METHOD line_line_angle : bool
VAR_INPUT
	p0:sc_pnt;
	p1:sc_pnt;
	p2:sc_pnt;
	angle_deg:REFERENCE TO LREAL;
END_VAR
VAR
	p00,p11,p22,v1,v2:Vector_3;
	dot,angle_rad:LREAL;
END_VAR
p00:=p_to_v(p0);
p11:=p_to_v(p1);
p22:=p_to_v(p2);

v1:=V3_SUB(p00,p11);
v2:=V3_SUB(p22,p11);

v1:=V3_NORMALIZED(v1);
v2:=V3_NORMALIZED(v2);

dot:=V3_DOT(v1,v2);
angle_rad:=ACOS(dot);
angle_deg:=angle_rad*to_degrees;
END_METHOD

METHOD arc_line_angle : bool
VAR_INPUT
	p0:sc_pnt;
	p1:sc_pnt;
	p2:sc_pnt;
	p3:sc_pnt;
	angle_deg:REFERENCE TO LREAL;
END_VAR
VAR
	pi:sc_pnt;

END_VAR
interpolate_arc(p0,p1,p2,0.9,pi);
line_line_angle(pi,p2,p3,angle_deg);
END_METHOD

METHOD p_to_v : Vector_3 //sc_pnt to vector3
VAR_INPUT
	in:sc_pnt;
END_VAR
p_to_v.x:=in.x;
p_to_v.y:=in.y;
p_to_v.z:=in.z;
END_METHOD

METHOD get_blockangles : BOOL
VAR_INPUT
	blockvec:REFERENCE TO vector_sc_segment;
	start:REFERENCE TO UDINT;
	end:REFERENCE TO UDINT;
END_VAR
VAR	
	i: UDINT;
	angle_deg:LREAL;
END_VAR
IF(blockvec.size()>0)THEN //! Vector safe.}
	
	FOR i:=start TO end-1 DO
		
		IF(blockvec.data[i].primitive_id=sc_primitive_id.line AND  blockvec.data[i+1].primitive_id=sc_primitive_id.line)THEN
			line_line_angle(blockvec.data[i].pnt_s,blockvec.data[i].pnt_e,blockvec.data[i+1].pnt_e,angle_deg);
			blockvec.data[i].angle_end:=angle_deg;
		END_IF
		
		IF(blockvec.data[i].primitive_id=sc_primitive_id.line AND (blockvec.data[i+1].primitive_id=sc_primitive_id.arc_ccw OR blockvec.data[i+1].primitive_id=sc_primitive_id.arc_cw))THEN
			line_arc_angle(blockvec.data[i].pnt_s,blockvec.data[i].pnt_e,blockvec.data[i+1].pnt_c,blockvec.data[i+1].pnt_e,angle_deg);
			blockvec.data[i].angle_end:=angle_deg;
		END_IF
		
		IF((blockvec.data[i].primitive_id=sc_primitive_id.arc_ccw OR blockvec.data[i].primitive_id=sc_primitive_id.arc_cw) AND blockvec.data[i+1].primitive_id=sc_primitive_id.line)THEN
			arc_line_angle(blockvec.data[i].pnt_s,blockvec.data[i].pnt_c,blockvec.data[i].pnt_e,blockvec.data[i+1].pnt_e,angle_deg);
			blockvec.data[i].angle_end:=angle_deg;
		END_IF
		
		IF((blockvec.data[i].primitive_id=sc_primitive_id.arc_ccw OR blockvec.data[i].primitive_id=sc_primitive_id.arc_cw) AND (blockvec.data[i+1].primitive_id=sc_primitive_id.arc_ccw OR blockvec.data[i+1].primitive_id=sc_primitive_id.arc_cw))THEN
			arc_arc_angle(blockvec.data[i].pnt_s,blockvec.data[i].pnt_c,blockvec.data[i].pnt_e,blockvec.data[i+1].pnt_c,blockvec.data[i+1].pnt_e,angle_deg);
			blockvec.data[i].angle_end:=angle_deg;
		END_IF
	END_FOR
END_IF
END_METHOD

METHOD get_corner_ve_blockangles : BOOL
VAR_INPUT
	blockvec:REFERENCE TO vector_sc_segment;
	start:REFERENCE TO UDINT;
	end:REFERENCE TO UDINT;
END_VAR
VAR	
	i: UDINT;
	angle_deg,factor,ve:LREAL;
END_VAR
IF(blockvec.size()<>0)THEN
	FOR i:=start TO  end-1 DO
		
		IF(blockvec.data[i].angle_end<=STOP_ANGLE)THEN //! Stop required.
			blockvec.data[i].vel_end:=0;
			//! Set next block vo to zero.
			IF(i<blockvec.size()-1)THEN
				blockvec.data[i+1].vel_start:=0;
			END_IF
		END_IF
	
		IF(blockvec.data[i].angle_end>STOP_ANGLE)THEN //! Percentage ve up to 180 degrees. //! 180 degrees = colinear.
			angle_deg:=blockvec.data[i].angle_end;
			factor:=(angle_deg-STOP_ANGLE)/STOP_ANGLE; //! 0-1, 1=straight on. 0=90 degrees.
			ve:=blockvec.data[i].vel_max*factor*ANGLE_VEL_FACTOR;
	
			blockvec.data[i].vel_end:=ve;
			//! Set next block vo to this ve.
			IF(i<blockvec.size()-1)THEN
				blockvec.data[i+1].vel_start:=ve;
			END_IF
		END_IF
		
	END_FOR
END_IF
END_METHOD

METHOD sc_get_gforce : bool
VAR_INPUT
	vel_mm_sec:LREAL;
	radius:LREAL;
	gforce:LREAL;
END_VAR
VAR	
	circumfence: LREAL;
	rps: LREAL;
	a:LREAL;
END_VAR
circumfence:=(radius*2)*M_PI;
rps:=vel_mm_sec/circumfence;
a:=4*(M_PI*M_PI)*radius*(rps*rps); //! [mm/s^2]
gforce:=a*0.0001; //! [g]
END_METHOD

METHOD get_velmax_gforce : bool
VAR_INPUT
	blockvec:REFERENCE TO vector_sc_segment;
	gforcemax:LREAL;
	start:REFERENCE TO UDINT;
	end:REFERENCE TO UDINT;
END_VAR
VAR
	i:UDINT;
	radius,gforce,maxvel_arc:LREAL;
	vm:LREAL;
END_VAR
IF(blockvec.size()<>0)THEN
	FOR i:=start TO end-1 DO
		IF(blockvec.data[i].primitive_id=sc_primitive_id.arc_cw OR blockvec.data[i].primitive_id=sc_primitive_id.arc_ccw)THEN	
			
			radius:=blockvec.data[i].radius;	
			
			//! Checks gforce using the program's velmax value.	
			vm:=blockvec.data[i].vel_max;							
			sc_get_gforce(vm,radius,gforce);
	
			IF(gforce>gforcemax)THEN
				maxvel_arc:=0;
				sc_set_gforce(radius,gforcemax,maxvel_arc);
				blockvec.data[i].vel_max:=maxvel_arc;
			END_IF			
		END_IF
	END_FOR
END_IF
END_METHOD

METHOD sc_optimize_all : BOOL
VAR_INPUT
	blockvec:REFERENCE TO vector_sc_segment;
	line_start:UDINT;
	line_end:UDINT;
END_VAR
line_start:=LIMIT(0,line_start,blockvec.size());
line_end:=LIMIT(line_start,line_end,blockvec.size());



//! Calculate motion block corners.
get_blockangles(blockvec,line_start,line_end);

//! Set end velocity, based on block corners, if no angle, ve is set to vm at this stage.
get_corner_ve_blockangles(blockvec,line_start,line_end);

//! Set the velmax for arc's using gforce value. Set the velmax for lines to program velmax.
get_velmax_gforce(blockvec,gforcemax,line_start,line_end);

//set g0 ve vo
sc_optimize_G0_ve(blockvec,line_start,line_end);

//optimize ve <--
sc_optimize_G123_ve_backward(blockvec,line_start,line_end);

//optimize ve -->
sc_optimize_G123_ve_forward(blockvec,line_start,line_end);
END_METHOD

METHOD sc_optimize_G0_ve : BOOL
VAR_INPUT
	blockvec:REFERENCE TO vector_sc_segment;
	start:REFERENCE TO UDINT;
	end:REFERENCE TO UDINT;
END_VAR
VAR
	i:UDINT;
END_VAR
IF(blockvec.size()<>0)THEN
	FOR i:=start TO end-1 DO
	
		//! End velocity=0 if motion is G0, rapid.
		IF(blockvec.data[i].primitive_id=sc_primitive_id.rapid)THEN 
			blockvec.data[i].vel_start:=0;
			blockvec.data[i].vel_end:=0;
	
			//! Set next block vo to 0.
			IF(i<blockvec.size()-1)THEN
				blockvec.data[i+1].vel_start:=0;
			END_IF
		END_IF
	END_FOR
END_IF
END_METHOD

METHOD sc_optimize_G123_ve_backward :BOOL
VAR_INPUT
	blockvec:REFERENCE TO vector_sc_segment;
	start:REFERENCE TO UDINT;
	end:REFERENCE TO UDINT;
END_VAR
VAR
	i:UDINT;
	vo,ve,vm,tarpos:LREAL;
	r_vel,r_acc,r_pos:LREAL;
	finish:BOOL;
	p_data:sc_data;
	pcurve:sc_engine;
	j:LREAL;
	
END_VAR
IF(blockvec.size()<>0)THEN
	FOR i:=end-1 TO start+1 BY-1 DO 
		
		IF(blockvec.data[i].primitive_id<>sc_primitive_id.rapid AND blockvec.data[i].primitive_id<>sc_primitive_id.empty)THEN 
			//! Swap vo,ve.
			ve:=blockvec.data[i].vel_start;
			vo:=blockvec.data[i].vel_end;
			vm:=blockvec.data[i].vel_max;
			tarpos:=blockvec.data[i].path_lenght;	

			MEMUtils.MemSet(ADR(p_data),0,SIZEOF(p_data));
			
			pcurve.set_cycle_time(CT,p_data);
			
			finish:=FALSE;
			WHILE NOT finish DO				
				pcurve.set_data(tarpos,vo,ve,vm,limits.max_acc,limits.max_jerk,1,p_data);	
				pcurve.update(p_data,1);
				pcurve.get_result(r_pos,r_vel,r_acc,finish,p_data);			
			END_WHILE
			
			IF(ve<>0)THEN
				blockvec.data[i].vel_start:=r_vel;
				blockvec.data[i-1].vel_end:=r_vel;
			END_IF
			
			blockvec.data[i].back_optim:=TRUE;
		END_IF
	END_FOR
END_IF
END_METHOD

METHOD sc_optimize_G123_ve_forward : BOOL
VAR_INPUT
	blockvec:REFERENCE TO vector_sc_segment;
	start:REFERENCE TO UDINT;
	end:REFERENCE TO UDINT;
END_VAR
VAR
	i:UDINT;
	vo,ve,vm,tarpos:LREAL;
	r_vel,r_acc,r_pos:LREAL;
	finish:BOOL;
	p_data:sc_data;
	pcurve:sc_engine;

END_VAR
IF(blockvec.size()<>0)THEN	
	FOR i:=start TO end-1 DO 
	
		IF(blockvec.data[i].primitive_id<>sc_primitive_id.rapid AND blockvec.data[i].primitive_id<>sc_primitive_id.empty)THEN 
	
			vo:=blockvec.data[i].vel_start;
			ve:=blockvec.data[i].vel_end;
			vm:=blockvec.data[i].vel_max;
			tarpos:=blockvec.data[i].path_lenght;
			
			MEMUtils.MemSet(ADR(p_data),0,SIZEOF(p_data));
			
			pcurve.set_cycle_time(CT,p_data);
						
			finish:=FALSE;
			WHILE NOT finish DO			
				pcurve.set_data(tarpos,vo,ve,vm,limits.max_acc,limits.max_jerk,1,p_data);	
				pcurve.update(p_data,1);
				pcurve.get_result(r_pos,r_vel,r_acc,finish,p_data);
			END_WHILE
			
			IF(ve<>0)THEN
				blockvec.data[i].vel_end:=r_vel;		
				IF(i<blockvec.size()-1)THEN  
					blockvec.data[i+1].vel_start:=r_vel;
				END_IF				
			END_IF
			
			blockvec.data[i].forward_optim:=TRUE;
		END_IF
	END_FOR
END_IF
END_METHOD

METHOD sc_set_gforce : bool
VAR_INPUT
	radius:LREAL;
	gforce:LREAL;
	vel_mm_sec:reference TO LREAL;
END_VAR

VAR
	rps: LREAL;
	circumfence: LREAL;
	a:LREAL;
END_VAR
circumfence:=(radius*2)*M_PI;
a:=gforce/0.0001;
rps:= SQRT(a/(4*(M_PI*M_PI)*radius));
vel_mm_sec:=rps*circumfence;
END_METHOD

METHOD interpolate_lenght
VAR_INPUT
	start,end,progress:LREAL;
	li:REFERENCE TO LREAL;
END_VAR
IF(start<end)THEN
	li:=start+(progress*NETTO(start,end));
	return;
END_IF
IF(start>end)THEN
	li:=start-(progress*NETTO(start,end));
	return;
END_IF
IF(start=end)THEN
	li:=end;
END_IF
END_METHOD

METHOD interpolate_arc
VAR_INPUT
	p1:sc_pnt;//! start position
	p2:sc_pnt;//! end position 
	center:sc_pnt;//! center IJK
	progress:LREAL;
	pi:REFERENCE TO sc_pnt;
END_VAR
VAR
	radius:LREAL;
	circumference:LREAL;
	startingAngle,endingAngle:LREAL;
	chordSquared,tau,chordHeight:LREAL;
	theta:LREAL;
	arcLengthMM:LREAL;
	angleNow:LREAL;

END_VAR
// add center offset IJ
center.x:=center.x+p1.x;
center.y:=center.y+p1.y;
// Compute geometry.
radius:=SQRT(EXPT(center.x-p1.x,2)+EXPT(center.y-p1.y,2)); 
circumference:=2.0*M_PI*radius;
startingAngle:=math.atan2(p1.y-center.y,p1.x-center.x);
endingAngle:=math.atan2(p2.y-center.y,p2.x-center.x);

// Compute chord height of arc.
chordSquared:=SQRT(EXPT(p2.x-p1.x,2)+EXPT(p2.y-p1.y,2));
tau:=SQRT(EXPT(radius,2)-(chordSquared/4));
chordHeight := radius - tau;

// Compute angle between lines.
theta:=endingAngle-startingAngle;

	//COUNTERCLOCKWISE
	IF (theta < 0)THEN
		theta:=theta+2*M_PI;
	END_IF

	//CLOCKWISE
	IF (theta >= 0)THEN	
		theta:=theta-2*M_PI;;
	END_IF


arcLengthMM:=ABS(circumference*(theta/(2*M_PI)));

//rotate point xy interpolate
angleNow:=startingAngle+theta*progress;
pi.x:=radius*COS(angleNow)+center.x;
pi.y:=radius*SIN(angleNow)+center.y;

IF(progress=1)THEN
	pi.x:=p2.x;
	pi.y:=p2.y;
END_IF

//z interpolate
interpolate_lenght(p1.z,p2.z,progress,pi.z);
END_METHOD

METHOD update_motion_and_interpolator : bool
VAR
	
END_VAR
//feed override
IF(pause_request OR stop_request)THEN
	maxvel_fo:=0;
ELSE
	maxvel_fo:=LIMIT(0,feed_override,100)/100;
END_IF


//motion cycle time
motion.set_cycle_time(CT,motion_data);

CASE state OF
	
	program_run://-------------------------------------------------------------------------------------------
	
		//motion
		motion.set_data(p.traject_lenght_end,p.vel_start,p.vel_end,p.vel_max,limits.max_acc,limits.max_jerk,maxvel_fo,motion_data);	
		motion.update(motion_data,0);
		motion.get_result(engine_outpos,velocity,acceleration,engine_finished,motion_data);
		//programmed vel
		programmed_velocity:=p.vel_max;
		
		//line progress
		line_progress:=(engine_outpos-p.traject_lenght_begin)/p.path_lenght;
		IF(FPU.IsLRealNaN(line_progress))THEN
			line_progress:=0;
		END_IF
		
		//interpolation
		IF(p.primitive_id=sc_primitive_id.line OR p.primitive_id=sc_primitive_id.rapid)THEN
			interpolate_line(p.pnt_s,p.pnt_e,line_progress,xyz);
		ELSIF(p.primitive_id=sc_primitive_id.arc_ccw OR p.primitive_id=sc_primitive_id.arc_cw)THEN
			interpolate_arc(p.pnt_s,p.pnt_e,p.pnt_c,line_progress,xyz);
		END_IF
		
	program_jog://-------------------------------------------------------------------------------------------
		
		
		motion.set_jog(jog_cmd.x_up,jog_cmd.x_dn,limits.min_quote_x,limits.max_quote_x,limits.max_vel,limits.max_acc,limits.max_jerk,motion_data);	
		motion.get_result(engine_outpos,velocity,acceleration,engine_finished,motion_data);
		xyz.x:=engine_outpos;
	
		
		
		
END_CASE
END_METHOD

METHOD interpolate_line
VAR_INPUT
	p0:sc_pnt;//! start point
	p1:sc_pnt;//! end pont
	progress:LREAL;
	pi:REFERENCE TO sc_pnt;
END_VAR
interpolate_lenght(p0.x,p1.x,progress,pi.x);
interpolate_lenght(p0.y,p1.y,progress,pi.y);
interpolate_lenght(p0.z,p1.z,progress,pi.z);
END_METHOD

METHOD round : LREAL
VAR_INPUT
	in : LREAL;
	N : INT;
END_VAR
VAR
	X: LREAL;
END_VAR
VAR
	DECADES : ARRAY[0..8] OF LREAL :=[ 1.0,10.0,100.0,1000.0,10000.0,10000.0,100000.0,1000000.0,10000000.0];
END_VAR
X := DECADES[LIMIT(0,N,8)];
ROUND := DINT_TO_LREAL(LREAL_TO_DINT(in * X)) / X;
END_METHOD

METHOD netto : LREAL
VAR_INPUT
	a,b:LREAL;
END_VAR
VAR
	diff_:LREAL;
END_VAR
diff_:=0;
IF(a<0 AND b<0)THEN
	a:=ABS(a);
	b:=ABS(b);
	diff_:=ABS(a-b);
END_IF
IF(a>=0 AND b>=0)THEN
	diff_:=ABS(a-b);
END_IF
IF(a<=0 AND b>=0)THEN
	diff_:=ABS(a)+b;
END_IF
IF(a>=0 AND b<=0)THEN
	diff_:=a+ABS(b);
END_IF
NETTO:=diff_;
END_METHOD

METHOD set_pnt_at : bool
VAR_INPUT
	pnt:REFERENCE TO sc_pnt;
	index:UDINT;
END_VAR
motion_vec.data[index].pnt_s:=pnt;
END_METHOD

END_FUNCTION_BLOCK

// MyController/Application/cnc/vector/functions/vector_at
FUNCTION vector_at : sc_segment
VAR_INPUT
	ptr:REFERENCE TO vector_sc_segment;
	index:UDINT;
END_VAR

IF(index>ptr.size()-1)THEN
	index:=ptr.size()-1;
END_IF
IF(index<0)THEN
	index:=0;
END_IF
vector_at:=ptr.data[index];

END_FUNCTION

// MyController/Application/cnc/vector/vector_sc_segment
FUNCTION_BLOCK vector_sc_segment
VAR_INPUT	
	data:ARRAY[0..MAX_GCODE_LINE+1]OF sc_segment;
END_VAR
VAR_OUTPUT
END_VAR
VAR	
	last_ptr:UDINT;
END_VAR

METHOD clear : bool
VAR_INPUT
END_VAR
VAR
	i:UDINT;
END_VAR
MEMUtils.MemSet(ADR(data),0,SIZEOF(data));
last_ptr:=0;
END_METHOD

METHOD end : UDINT
VAR_INPUT
END_VAR
end:=last_ptr;
END_METHOD

METHOD begin : int
VAR_INPUT
END_VAR
begin:=0;
END_METHOD

METHOD push_back : bool
VAR_INPUT
	in:sc_segment;
END_VAR
MEMUtils.MemCpy(ADR(data[last_ptr]),ADR(in),SIZEOF(in));
last_ptr:=last_ptr+1;
END_METHOD

METHOD back : sc_segment
VAR_INPUT
END_VAR
back:=data[last_ptr-1];
END_METHOD

METHOD front : sc_segment
VAR_INPUT
END_VAR
front:=data[0];
END_METHOD

METHOD size : UDINT
VAR_INPUT
END_VAR
size:=last_ptr;
END_METHOD

METHOD insert : bool
VAR_INPUT
	pos:UDINT;
	vec:REFERENCE TO vector_sc_segment;
END_VAR
VAR
	i:UDINT;
END_VAR
//libero lo spazio spostando avanti i vettori successivi al punto di inserimento
IF(vec.size()>0)THEN
	IF(last_ptr<>0)THEN
		FOR i:=pos TO last_ptr-1 DO
			MEMUtils.MemCpy(ADR(data[i+vec.size()]),ADR(data[i]),SIZEOF(data[i]));
			//data[i+vec.size()]:=data[i];
		END_FOR
		last_ptr:=i+vec.size();
	END_IF


	//copio il nuovo array partendo dalla posizione desiderata
	FOR i:=0 TO vec.size()-1 DO
		MEMUtils.MemCpy(ADR(data[i+pos]),ADR(vec.data[i]),SIZEOF(vec.data[i]));
		//data[i+pos]:=vec.data[i];
		//se non ho inserito prima nessun vettore,avanzo il puntatore alla fine della lunghezza del vettore che copio
		IF(last_ptr=0)THEN
			last_ptr:=i+vec.size();
		END_IF 	
	END_FOR
END_IF
END_METHOD

END_FUNCTION_BLOCK

// MyController/Application/cnc/vector/functions/vector_nr_increment
FUNCTION vector_nr_increment : bool
VAR_INPUT
	ptr:REFERENCE TO vector_sc_segment;
	n:REFERENCE TO UDINT;
END_VAR

n:=n+1;
n:=MIN(n,ptr.size());
n:=MAX(n,0);

END_FUNCTION

// MyController/Application/cnc/motion/sc_engine
FUNCTION_BLOCK sc_engine
VAR_INPUT
END_VAR
VAR_OUTPUT
END_VAR
VAR
END_VAR

METHOD set_data : bool
VAR_INPUT
	ds:LREAL;//target
	vo:LREAL;//begin velocity
	ve:LREAL;//end velocity
	vs:LREAL;//max velocity
	a:LREAL;//acceleration
	gain:LREAL;//0-100
	ovr:LREAL;//override 0-1
	p:REFERENCE TO sc_data;//data structure
END_VAR
//!limit gain
gain:=LIMIT(0.001,gain,100);

ve:=ve*ovr;
vs:=vs*ovr;

IF(vs=0)THEN
	vs:=0.000001;
	p.stop:=TRUE;
END_IF

//target position change
IF(ds<>p.ds_old)THEN
	p.ds:=ds;
	p.ds_old:=p.ds;
	p.init:=TRUE;
END_IF

//max vel change
IF(vs<>p.vs_old)THEN
	p.vs:=vs;
	p.vs_old:=p.vs;
	p.init:=TRUE;
END_IF

p.vo:=vo;
p.vs:=vs;
p.ve:=ve;
p.a:=a;
p.gain:=gain;
END_METHOD

METHOD get_result : bool
VAR_INPUT
	pos:REFERENCE TO LREAL;
	vel:REFERENCE TO LREAL;
	acc:REFERENCE TO LREAL;
	finish:REFERENCE TO BOOL;
	p:REFERENCE TO sc_data;
END_VAR
pos:=p.sc_sr_inc;
vel:=p.sc_vr*p.dir;
acc:=p.sc_ar*p.dir;
finish:=p.finish;
END_METHOD

METHOD set_cycle_time : bool
VAR_INPUT
	t:LREAL;
	p:reference TO sc_data;
END_VAR
p.cycle_time:=t;
END_METHOD

METHOD update
VAR_INPUT
	p:REFERENCE TO sc_data;
	use_vo:BOOL;
END_VAR
//new movement request
IF(p.init)THEN
	p.finish:=FALSE;
	p.init:=FALSE;
	//direction
	IF(p.ds>=p.sc_sr_inc)THEN
		p.dir:=1;
	END_IF
	IF(p.ds<p.sc_sr_inc)THEN
		p.dir:=-1;
	END_IF
	//targets
	p.t_pos:=ABS(p.sc_sr_inc-p.ds);
	IF(NOT use_vo)THEN
		p.t_vin:=p.sc_vr;
	ELSE
		p.t_vin:=p.vo;
	END_IF		
	//store position to old position
	p.sc_sr_inc_old:=p.sc_sr_inc;
	//zero timer
	p.at_time:=0;
END_IF

//process curve 
motion(p.t_pos,p.t_vin,p.ve,p.vs,p.a,p.gain,p);

//inc position
p.sc_sr_inc:=p.sc_sr_inc_old+(p.sc_sr*p.dir);

//check finish
IF(p.at_time+p.cycle_time>=p.tr_ct)THEN	
	p.sc_sr_inc:=p.ds;
	p.finish:=TRUE;	
	p.state:=sc_motion_status.motion_finish;
	RETURN;	
END_IF

//if stop and vel c=0 ... stop time increment ... motion not finished ... 
IF(p.stop AND p.sc_vr<=0.1)THEN
	p.stop:=FALSE;
	p.sc_ar:=0;
	p.sc_vr:=0;
	p.state:=sc_motion_status.motion_pause;	
ELSE	
	//time increment.. normal condition..
	p.at_time:=p.at_time+p.cycle_time;
	p.state:=sc_motion_status.motion_process;
END_IF
END_METHOD

METHOD motion : BOOL
VAR_INPUT
	ds:LREAL;//target
	vo:LREAL;//begin velocity
	ve:LREAL;//end velocity
	vs:LREAL;//max velocity
	a:LREAL;//acceleration
	gain:LREAL;//0-100
	p:REFERENCE TO sc_data;//data structure
END_VAR
VAR
	t1,t2,t3,s1,s2,s3,v1,ct,cs,vr,sr,ar,t:LREAL;
	prompt_new_ve:BOOL;
	res:sc_data;
END_VAR

//! ds=displacement.
//! vo=velocity begin.
//! ve=velocity end.
//! vs=velocity max.
//! a=acceleration.
//! at_time=request at timestamp.
//! gain=curve power.

//! Traditional lineair curve
t1:=0;
t2:=0;
t3:=0;
s1:=0;
s2:=0;
s3:=0;
v1:=0;
ct:=0;
cs:=0;
vr:=0;
sr:=0;
ar:=0;
t:=p.at_time;

//! formula's lineair acceleration:
//! v*v=(vo*vo) + 2*a*ds, ds=vo*t + 0.5*a*(t*t), t=sqrt(s*2/a) ,v=vo+a*t
//! formula's lineair steady:
//! s=vo+ v*t, t=s/v
//! formula's scurve:
//! a(t)=jm*t
//! v(t)=vo+jm*(t*t)/2
//! ds(t)=vo*t+jm*(t*t*t)/6


//! Curve steady algo.
IF(vo=ve AND vo=vs)THEN
	res.sc_vr:=ve;
	res.tr_ct:=ds/ve;
	res.tr_cs:=ds;
	res.sc_ar:=0;
	//res.sc_sr:=vo+ ve*t;
	res.sc_sr:=ve*t;
	p.sc_ct:=res.sc_ct;
	p.sc_jm:=res.sc_jm;
	p.sc_cs:=res.sc_cs;
	p.sc_vr:=res.sc_vr;
	p.sc_sr:=res.sc_sr;
	p.sc_ar:=res.sc_ar;
	p.tr_ct:=res.tr_ct;
	p.tr_cs:=res.tr_cs;
	RETURN;
END_IF

//! Curve down algo.
// if(ve<vo && vs>0 && s>0)
 IF(vo>=vs AND vs>=ve AND vs>0 AND ds>0)THEN

	//! Limits
	IF(vs>vo)THEN
		vs:=vo;
	END_IF
	IF(ve>vs)THEN
		ve:=vs;
	END_IF

	//! Dcc period to vs.
	res:=Sc_bck(gain,a,vo,vs,0);
	t1:=res.sc_ct;
	s1:=res.sc_cs;

	//! Dcc vs to ve period.
	res:=Sc_bck(gain,a,vs,ve,0);
	t3:=res.sc_ct;
	s3:=res.sc_cs;

	//! Vs steady period.
	s2:=ds-(s1+s3);
	t2:=s2/vs;

	prompt_new_ve:=0;
	IF(t2<0)THEN //! Ve can not be reached. Set new ve based on s.

		ve:=SQRT((vo*vo) + 2*-a*ds);
		t1:=(vo-ve)/a;
		s1:=ABS(vo*t1 +0.5*-a*(t1*t1));

		t2:=0; //! Only t1 is used in this case.
		t3:=0;
		s2:=0;
		s3:=0;

		prompt_new_ve:=1;
	END_IF

	res:=Sc_bck(gain,a,vo,vs,t1);
	v1:=res.sc_vr;

	ct:=t1+t2+t3;
	cs:=s1+s2+s3;
	res.tr_ct:=ct;
	res.tr_cs:=cs;

	IF(t<t1)THEN //! Period 1.
		IF(prompt_new_ve)THEN
			res:=Sc_bck(100,a,vo,ve,t); //! 100=gain
			res.tr_ct:=ct;
			res.tr_cs:=cs;
			p.sc_ct:=res.sc_ct;
			p.sc_jm:=res.sc_jm;
			p.sc_cs:=res.sc_cs;
			p.sc_vr:=res.sc_vr;
			p.sc_sr:=res.sc_sr;
			p.sc_ar:=res.sc_ar;
			p.tr_ct:=res.tr_ct;
			p.tr_cs:=res.tr_cs;
			RETURN;
		END_IF
		res:=Sc_bck(gain,a,vo,vs,t);
		res.tr_ct:=ct;
		res.tr_cs:=cs;
		p.sc_ct:=res.sc_ct;
		p.sc_jm:=res.sc_jm;
		p.sc_cs:=res.sc_cs;
		p.sc_vr:=res.sc_vr;
		p.sc_sr:=res.sc_sr;
		p.sc_ar:=res.sc_ar;
		p.tr_ct:=res.tr_ct;
		p.tr_cs:=res.tr_cs;
		RETURN;
	END_IF
	IF(t>=t1 AND t<=t1+t2)THEN //! Period 2.
		t:=t-t1;

		IF(t1=0)THEN
			v1:=vo;
		END_IF

		res.sc_vr:=v1;
		res.sc_sr:=s1 + (v1*t);
		res.sc_ar:=0;
		res.tr_ct:=ct;
		res.tr_cs:=cs;
		p.sc_ct:=res.sc_ct;
		p.sc_jm:=res.sc_jm;
		p.sc_cs:=res.sc_cs;
		p.sc_vr:=res.sc_vr;
		p.sc_sr:=res.sc_sr;
		p.sc_ar:=res.sc_ar;
		p.tr_ct:=res.tr_ct;
		p.tr_cs:=res.tr_cs;
		RETURN;
	END_IF
	IF(t>t1+t2)THEN //! Period 3.
		t:=t-t1;
		t:=t-t2;

		res:=Sc_bck(gain,a,vs,ve,t);
		res.sc_sr:=res.sc_sr+s1;
		res.sc_sr:=res.sc_sr+s2;
		res.tr_ct:=ct;
		res.tr_cs:=cs;
		p.sc_ct:=res.sc_ct;
		p.sc_jm:=res.sc_jm;
		p.sc_cs:=res.sc_cs;
		p.sc_vr:=res.sc_vr;
		p.sc_sr:=res.sc_sr;
		p.sc_ar:=res.sc_ar;
		p.tr_ct:=res.tr_ct;
		p.tr_cs:=res.tr_cs;
		RETURN;
	END_IF
END_IF

//! Curve up algo.
//if(ve>=vo && vs>0 && ds>0){
IF(vo<=vs AND vs>0 AND ds>0)THEN

	//! Limits.
	IF(ve>vs)THEN	
		ve:=vs;
	END_IF

	res:=Sc_fwd(gain,a,vo,ve,0.0);
	t1:=res.sc_ct;
	s1:=res.sc_cs;

	prompt_new_ve:=0;
	IF(s1>ds)THEN //! Ve can not be reached! Set new ve based on ds.
		t1:=SQRT(ds/(0.5*a));
		ve:=vo+a*t1;

		res.sc_ct:=t1;
		res.sc_cs:=ds;

		vr:=vo+a*t;
		sr:=0.5*a*(t*t);
		ar:=a;

		prompt_new_ve:=1;
	END_IF

	//! Sample to fit.
	WHILE(1)DO

		//! Acc period.
		res:=Sc_fwd(gain,a,vo,vs,0.0);
		t1:=res.sc_ct;
		s1:=res.sc_cs;
		IF(t1<0)THEN
			t1:=0;
		END_IF

		//! Dcc period.
		res:=Sc_bck(gain,a,vs,ve,0.0);
		t3:=res.sc_ct;
		s3:=res.sc_cs;
		IF(t3<0)THEN
			t3:=0;
		END_IF

		//! Steady period.
		s2:=ds-(s1+s3);
		t2:=s2/vs;

		IF(s1+s3<=ds)THEN
			EXIT;
		ELSE 
			vs:=vs-0.01*vs;	//! Important value. It reduces mavel by input value until curves fit.
							//! The reduce value has great impact on function cycle time.
							//! 0.1 = 10% velocity recude to find the fit.
		END_IF
	END_WHILE

	res:=Sc_fwd(gain,a,vo,vs,t1);
	v1:=res.sc_vr;

	ct:=t1+t2+t3;
	cs:=s1+s2+s3;
	res.tr_ct:=ct;
	res.tr_cs:=cs;

	IF(t<t1)THEN //! Period 1.
		IF(prompt_new_ve)THEN
			res:=Sc_fwd(100.0,a,vo,ve,t);
			res.tr_ct:=ct;
			res.tr_cs:=cs;
			p.sc_ct:=res.sc_ct;
			p.sc_jm:=res.sc_jm;
			p.sc_cs:=res.sc_cs;
			p.sc_vr:=res.sc_vr;
			p.sc_sr:=res.sc_sr;
			p.sc_ar:=res.sc_ar;
			p.tr_ct:=res.tr_ct;
			p.tr_cs:=res.tr_cs;
			RETURN;
		END_IF

		res:=Sc_fwd(gain,a,vo,vs,t);
		res.tr_ct:=ct;
		res.tr_cs:=cs;
		p.sc_ct:=res.sc_ct;
		p.sc_jm:=res.sc_jm;
		p.sc_cs:=res.sc_cs;
		p.sc_vr:=res.sc_vr;
		p.sc_sr:=res.sc_sr;
		p.sc_ar:=res.sc_ar;
		p.tr_ct:=res.tr_ct;
		p.tr_cs:=res.tr_cs;
		RETURN;
	END_IF
	IF(t>=t1 AND t<=t1+t2)THEN //! Period 2.
		t:=t-t1;

		res.sc_vr:=v1;
		res.sc_sr:=s1 + (v1*t);
		res.sc_ar:=0;
		res.tr_ct:=ct;
		res.tr_cs:=cs;
		p.sc_ct:=res.sc_ct;
		p.sc_jm:=res.sc_jm;
		p.sc_cs:=res.sc_cs;
		p.sc_vr:=res.sc_vr;
		p.sc_sr:=res.sc_sr;
		p.sc_ar:=res.sc_ar;
		p.tr_ct:=res.tr_ct;
		p.tr_cs:=res.tr_cs;
		RETURN;
	END_IF
	IF(t>t1+t2 AND t<=t1+t2+t3)THEN //! Period 3.
		t:=t-t1;
		t:=t-t2;

		res:=Sc_bck(gain,a,vs,ve,t);
		res.sc_sr:=res.sc_sr+s1;
		res.sc_sr:=res.sc_sr+s2;
		res.tr_ct:=ct;
		res.tr_cs:=cs;
		p.sc_ct:=res.sc_ct;
		p.sc_jm:=res.sc_jm;
		p.sc_cs:=res.sc_cs;
		p.sc_vr:=res.sc_vr;
		p.sc_sr:=res.sc_sr;
		p.sc_ar:=res.sc_ar;
		p.tr_ct:=res.tr_ct;
		p.tr_cs:=res.tr_cs;
		RETURN;
	END_IF
END_IF


p.sc_ct:=res.sc_ct;
p.sc_jm:=res.sc_jm;
p.sc_cs:=res.sc_cs;
p.sc_vr:=res.sc_vr;
p.sc_sr:=res.sc_sr;
p.sc_ar:=res.sc_ar;
p.tr_ct:=res.tr_ct;
p.tr_cs:=res.tr_cs;
END_METHOD

METHOD Sc_bck : sc_data
VAR_INPUT
	gain:LREAL;//curve power
	am:LREAL;//acceleration
	vo:LREAL;//begin velocity
	ve:LREAL;//end velocity
	at_time:LREAL;//request curve state at timestamp[t]
END_VAR
VAR
	res:sc_data;
	vo_temp,as,jm,v1,v2,v3,s1,s2,s3,t1,t2,t3,t:LREAL;
END_VAR

//! Invert vo,ve
vo_temp:=vo;
vo:=ve;
ve:=vo_temp;

//! formula's lineair acceleration:
//! v*v=(vo*vo) + 2*a*s, s=vo*t + 0.5*a*(t*t), t=sqrt(s*2/a) ,v=vo+a*t
//! formula's lineair steady:
//! s=vo+ v*t, t=s/v
//! formula's scurve:
//! a(t)=jm*t
//! v(t)=vo+jm*(t*t)/2
//! s(t)=vo*t+jm*(t*t*t)/6

//! Calculated acc at inflection point.
as:=0;
//! Jerk.
jm:=0;
//! Velocity.
v1:=0;
v2:=0;
v3:=0;
//! Displacement.
s1:=0;
s2:=0;
s3:=0;
//! Periods. t1=concave, t2=lineair transition, t3=convex.
t1:=0;
t2:=0;
t3:=0;

//! Gain 0-100% to make it more user friendly.
//!
//! 100% gain is full scurve without lineair transition period.
//! 0.001% gain is a traditional lineair curve.
gain:=gain*((ve-vo)/100);
gain:=MAX(gain,0.001);

as:=2*am;
t1:=gain/as;
jm:=as/t1;
t3:=t1;



//! Calculate period t2. Here we use no vo values.
v1:=0 +jm*(t1*t1)/2;                 //! Velocity end has priority.
v3:=v1;
v2:=(ve-vo)-(v1+v3);
t2:=v2/as;

//! Totals, used by t<. requests below.
IF(t2<0)THEN
	t2:=0;
END_IF
IF(t2>0)THEN                          //! Gain value = < ve-vo.
	v1:=vo +jm*(t1*t1)/2;
	v2:=v1+as*t2;
	v3:=v2 + as*t3 - jm*(t3*t3)/2;

	s1:=vo*t1 +jm*(t1*t1*t1)/6;
	s2:=s1+ v1*t2+0.5*as*(t2*t2);
	s3:=s2+ v2*t3 + as*(t3*t3)/2 - jm*(t3*t3*t3)/6;
END_IF
IF(t2=0)THEN                          //! Gain value = ~(ve-vo).
	v1:=vo +jm*(t1*t1)/2;
	v2:=0;
	v3:=v1 + as*t3 - jm*(t3*t3)/2;

	s1:=vo*t1 +jm*(t1*t1*t1)/6;
	s2:=0;
	s3:=s1+ v1*t3 + as*(t3*t3)/2 - jm*(t3*t3*t3)/6;
END_IF

res.sc_ct:=t1+t2+t3;                        //! Total curve time.

IF(fpu.IsLRealNaN(res.sc_ct))THEN
	res.sc_ct:=0;
END_IF
res.sc_cs:=s3;

//! Invert time.
t:=res.sc_ct-at_time;

IF(t<t1)THEN                           //! Period concave t1
	v1:=vo +jm*(t*t)/2;
	s1:=vo*t +jm*(t*t*t)/6;

	res.sc_vr:=v1;
	res.sc_sr:=res.sc_cs-s1;             //! Invert displacement.
	res.sc_ar:=-ABS(jm*t);        //! Invert acceleration.
	Sc_bck := res;
	RETURN;
END_IF
IF(t>=t1 AND t<=t1+t2)THEN              //! Period lineair transition t2
	t:=t - t1;
	v2:=v1+as*t;
	s2:=s1+ v1*t+0.5*as*(t*t);

	res.sc_vr:=v2;
	res.sc_sr:=res.sc_cs-s2;             //! Invert displacement.
	res.sc_ar:=-ABS(as);          //! Invert acceleration.
	Sc_bck := res;
	RETURN;
END_IF
IF(t>t1+t2 AND t<=t1+t2+t3)THEN          //! Period convex t3
	t:=t-t1;
	t:=t-t2;

	IF(t2=0)THEN
		v2:=v1;
		s2:=s1;
	END_IF

	v3:=v2 + as*t - jm*(t*t)/2;
	s3:=s2+ v2*t + as*(t*t)/2 - jm*(t*t*t)/6;

	res.sc_vr:=v3;
	res.sc_sr:=res.sc_cs-s3;             //! Invert displacement.
	res.sc_ar:=-ABS(as-jm*t);     //! Invert acceleration.
	Sc_bck := res;
	RETURN;
END_IF

//! Normally don't get here.
Sc_bck := res;
END_METHOD

METHOD Sc_fwd : sc_data
VAR_INPUT
	gain:LREAL;//curve power
	am:LREAL;//acceleration
	vo:LREAL;//begin velocity
	ve:LREAL;//end velocity
	at_time:LREAL;//request curve state at timestamp[t]
END_VAR
VAR
	res:Sc_data;
	as,jm,v1,v2,v3,s1,s2,s3,t,t1,t2,t3:LREAL;
END_VAR
//! formula's lineair acceleration:
//! v*v=(vo*vo) + 2*a*s, s=vo*t + 0.5*a*(t*t), t=sqrt(s*2/a) ,v=vo+a*t
//! formula's lineair steady:
//! s=vo+ v*t, t=s/v
//! formula's scurve:
//! a(t)=jm*t
//! v(t)=vo+jm*(t*t)/2
//! s(t)=vo*t+jm*(t*t*t)/6

//! Calculated acc at inflection point.
as:=0;
//! Jerk.
jm:=0;
//! Velocity.
v1:=0;
v2:=0;
v3:=0;
//! Displacement.
s1:=0;
s2:=0;
s3:=0;
//! Periods. t1=concave, t2=lineair transition, t3=convex.
t1:=0;
t2:=0;
t3:=0;

//! Gain 0-100% to make it more user friendly.
//!
//! 100% gain is full scurve without lineair transition period.
//! 0.001% gain is a traditional lineair curve.
gain:=gain*((ve-vo)/100);
gain:=MAX(gain,0.001);

as:=2*am;
t1:=gain/as;
jm:=as/t1;
t3:=t1;



//! Calculate period t2. Here we use no vo values.
v1:=0 +jm*(t1*t1)/2;                 //! Velocity end has priority.
v3:=v1;
v2:=(ve-vo)-(v1+v3);
t2:=v2/as;

//! Totals, used by [t<..] requests below.
IF(t2<0)THEN
	t2:=0;
END_IF

IF(t2>0)THEN                          //! Gain value = < ve-vo.
	v1:=vo +jm*(t1*t1)/2;
	v2:=v1+as*t2;
	v3:=v2 + as*t3 - jm*(t3*t3)/2;

	s1:=vo*t1 +jm*(t1*t1*t1)/6;
	s2:=s1+ v1*t2+0.5*as*(t2*t2);
	s3:=s2+ v2*t3 + as*(t3*t3)/2 - jm*(t3*t3*t3)/6;
END_IF
IF(t2=0)THEN                          //! Gain value = ~(ve-vo).
	v1:=vo +jm*(t1*t1)/2;
	v2:=0;
	v3:=v1 + as*t3 - jm*(t3*t3)/2;

	s1:=vo*t1 +jm*(t1*t1*t1)/6;
	s2:=0;
	s3:=s1+ v1*t3 + as*(t3*t3)/2 - jm*(t3*t3*t3)/6;
END_IF

res.sc_ct:=t1+t2+t3;                        //! Total curve time.
IF(fpu.IsLRealNaN(res.sc_ct))THEN
	res.sc_ct:=0;
END_IF
res.sc_cs:=s3;

t:=at_time;

IF(t<t1)THEN                         //! Period concave t1
	v1:=vo +jm*(t*t)/2;
	s1:=vo*t +jm*(t*t*t)/6;

	res.sc_vr:=v1;
	res.sc_sr:=s1;
	res.sc_ar:=jm*t;
	Sc_fwd := res;
	RETURN;
END_IF
IF(t>=t1 AND t<=t1+t2)THEN              //! Period lineair transition t2}
	t:=t-t1;
	v2:=v1+as*t;
	s2:=s1+ v1*t+0.5*as*(t*t);

	res.sc_vr:=v2;
	res.sc_sr:=s2;
	res.sc_ar:=as;
	Sc_fwd := res;
	RETURN;
END_IF
IF(t>t1+t2 AND t<=t1+t2+t3)THEN          //! Period convex t3
	t:=t-t1;
	t:=t-t2;

	IF(t2=0)THEN
		v2:=v1;
		s2:=s1;
	END_IF

	v3:=v2 + as*t - jm*(t*t)/2;
	s3:=s2+ v2*t + as*(t*t)/2 - jm*(t*t*t)/6;

	res.sc_vr:=v3;
	res.sc_sr:=s3;
	res.sc_ar:=as-jm*t;
	Sc_fwd := res;
	RETURN;
END_IF

//! Normally don't get here.
Sc_fwd := res;
END_METHOD

METHOD get_status : sc_motion_status
VAR_INPUT
	p:REFERENCE TO sc_data;
END_VAR
get_status:=p.state;
END_METHOD

METHOD set_pos : bool
VAR_INPUT
	pos:LREAL;
	p:REFERENCE TO sc_data;//data structure
END_VAR
p.sc_sr_inc:=p.sc_sr_inc_old:=pos;
END_METHOD

METHOD set_jog : bool
VAR_INPUT
	fwd:BOOL;
	rev:BOOL;
	min_pos:LREAL;
	max_pos:LREAL;
	vs:LREAL;//max velocity
	a:LREAL;//acceleration
	gain:LREAL;//0-100
	p:REFERENCE TO sc_data;//data structure
END_VAR

VAR
	r_vel,r_acc,r_pos:LREAL;
	finish:BOOL;
END_VAR
IF(fwd)THEN
	p.jog_fwd:=fwd;
	p.jog_rev:=FALSE;
END_IF
IF(rev)THEN
	p.jog_fwd:=FALSE;
	p.jog_rev:=rev;
END_IF

//!limit gain
gain:=LIMIT(0.001,gain,100);

IF(vs=0)THEN
	vs:=0.000001;
END_IF

IF(p.jog_fwd)THEN
	p.ds:=max_pos;
END_IF
IF(p.jog_rev)THEN
	p.ds:=min_pos;
END_IF
IF(p.ds<>p.ds_old)THEN
	p.ds_old:=p.ds;
	p.init:=TRUE;
END_IF

//max vel change
IF(vs<>p.vs_old)THEN
	p.vs:=vs;
	p.vs_old:=p.vs;
	p.init:=TRUE;
END_IF

p.vo:=0;
p.vs:=vs;
p.ve:=0;
p.a:=a;
p.gain:=gain;


//-------------------------------------------------------


//check inversion on fly ....with velocity <>0
get_result(r_pos,r_vel,r_acc,finish,p);
IF((p.jog_fwd AND r_vel<0) OR (p.jog_rev AND r_vel>0))THEN
	p.vs:=0.000001;
	p.init:=TRUE;
	p.stop:=TRUE;
END_IF

//new movement request
IF(p.init)THEN
	p.finish:=FALSE;
	p.init:=FALSE;		
	//direction
	IF(p.ds>=p.sc_sr_inc)THEN
		p.dir:=1;
	END_IF
	IF(p.ds<p.sc_sr_inc)THEN
		p.dir:=-1;
	END_IF
	//targets
	p.t_pos:=ABS(p.sc_sr_inc-p.ds);
	p.t_vin:=p.sc_vr;	
	//store position to old position
	p.sc_sr_inc_old:=p.sc_sr_inc;
	//zero timer
	p.at_time:=0;
END_IF

//process curve 
motion(p.t_pos,p.t_vin,0,p.vs,p.a,p.gain,p);

//inc position
p.sc_sr_inc:=p.sc_sr_inc_old+(p.sc_sr*p.dir);

//check finish
IF(p.at_time+p.cycle_time>=p.tr_ct)THEN	
	p.sc_sr_inc:=p.ds;
	p.sc_ar:=0;
	p.sc_vr:=0;
	p.finish:=TRUE;	
	p.state:=sc_motion_status.motion_finish;
	RETURN;	
END_IF

//if stop and vel c=0 ... stop time increment ... motion not finished ... 
IF(p.stop AND p.sc_vr<=0.1)THEN
	p.stop:=FALSE;
	p.sc_ar:=0;
	p.sc_vr:=0;
	p.state:=sc_motion_status.motion_pause;	
ELSE	
	//time increment.. normal condition..
	p.at_time:=p.at_time+p.cycle_time;
	p.state:=sc_motion_status.motion_process;
END_IF
END_METHOD

METHOD jog_stop : bool
VAR_INPUT
	p:REFERENCE TO sc_data;//data structure
END_VAR

VAR
	
END_VAR
IF(p.sc_ar=0)THEN
	//stop curve to 0 vel
	motion(p.t_pos,p.sc_vr,0,0.00001,p.a,p.gain,p);	
ELSE
	//finish the last curve/2
	motion(p.t_pos,p.t_vin,0,p.vs,p.a,p.gain,p);
END_IF

//inc position
p.sc_sr_inc:=p.sc_sr_inc_old+(p.sc_sr*p.dir);

//time increment.. 
p.at_time:=p.at_time+p.cycle_time;
p.state:=sc_motion_status.motion_process;
END_METHOD

END_FUNCTION_BLOCK

// MyController/Application/cnc/vector/functions/round
FUNCTION round : lreal
VAR_INPUT
	in : LREAL;
	N : INT;
END_VAR
VAR
	X: LREAL;
END_VAR
VAR
	DECADES : ARRAY[0..8] OF LREAL :=[ 1.0,10.0,100.0,1000.0,10000.0,10000.0,100000.0,1000000.0,10000000.0];
END_VAR

X := DECADES[LIMIT(0,N,8)];
ROUND := DINT_TO_LREAL(LREAL_TO_DINT(in * X)) / X;

END_FUNCTION

// MyController/Application/cnc/vector3/V3_SUB
FUNCTION V3_SUB : vector_3//subtracts two vectors in a 3 dimensional space
VAR_INPUT
	A : Vector_3;
	B : Vector_3;
END_VAR

V3_SUB.X := A.X - B.X;
V3_SUB.Y := A.Y - B.Y;
V3_SUB.Z := A.Z - B.Z;

END_FUNCTION

// MyController/Application/cnc/vector3/V3_NORMALIZED
FUNCTION V3_NORMALIZED : vector_3
VAR_INPUT
	A : Vector_3;
END_VAR
VAR
	la: LREAL;
END_VAR

la := V3_ABS(A);
IF la > 0.0 THEN
	V3_NORMALIZED := V3_SMUL(A, 1.0 / la);
END_IF;

END_FUNCTION

// MyController/Application/cnc/vector3/V3_ABS
FUNCTION V3_ABS : LREAL
VAR_INPUT
	A : Vector_3;
END_VAR

V3_ABS := SQRT(A.X * A.X + A.Y * A.Y + A.Z * A.Z);

END_FUNCTION

// MyController/Application/cnc/vector3/V3_SMUL
FUNCTION V3_SMUL : vector_3//multiplies a vectors in a 3 dimensional space with a skalar M
VAR_INPUT
	A : Vector_3;
	M : LREAL;
END_VAR

V3_SMUL.X := A.X * M;
V3_SMUL.Y := A.Y * M;
V3_SMUL.Z := A.Z * M;

END_FUNCTION

// MyController/Application/cnc/vector3/V3_DOT
FUNCTION V3_DOT : LREAL
VAR_INPUT
	A : Vector_3;
	B : Vector_3;
END_VAR

V3_DOT := A.X * B.X + A.Y * B.Y + A.Z * B.Z;

END_FUNCTION

// MyController/Application/cnc/vector3/V3_ANG
FUNCTION V3_ANG : LREAL
VAR_INPUT
	A : Vector_3;
	B : Vector_3;
END_VAR
VAR
	d : LREAL;
END_VAR

d := V3_ABS(A) * V3_ABS(B);
IF d > 0 THEN
	V3_ANG := ACOS(LIMIT(-1.0, V3_DOT(A, B) / d,1.0));
END_IF;

END_FUNCTION

// MyController/Application/cnc/vector/functions/vector_traject_lenght
FUNCTION vector_traject_lenght : bool
VAR_INPUT
	ptr:REFERENCE TO  vector_sc_segment;
	l:REFERENCE TO LREAL;
END_VAR
VAR
	i:UDINT;
END_VAR

FOR i:=0 TO ptr.size()-1 DO
	l:=l+ptr.data[i].path_lenght;
END_FOR

END_FUNCTION

// MyController/Application/cnc/vector/functions/vector_nr_decrement
FUNCTION vector_nr_decrement : bool
VAR_INPUT
	ptr:REFERENCE TO vector_sc_segment;
	n:REFERENCE TO UDINT;
END_VAR

n:=n-1;
n:=MIN(n,ptr.size());
n:=MAX(n,0);

END_FUNCTION

// MyController/Application/cnc/vector3/V3_NUL
FUNCTION V3_NUL : BOOL
VAR_INPUT
	A : Vector_3;
END_VAR

V3_NUL := A.X = 0.0 AND A.Y = 0.0 AND A.Z = 0.0;

END_FUNCTION

// MyController/Application/cnc/vector3/V3_PAR
FUNCTION V3_PAR : BOOL//checks if two vectors in a 3 dimensional space are parallel
VAR_INPUT
	A : Vector_3;
	B : Vector_3;
END_VAR

V3_PAR := V3_ABS(V3_CROSS(A, B)) = 0.0;

END_FUNCTION

// MyController/Application/cnc/vector3/V3_CROSS
FUNCTION V3_CROSS : vector_3
VAR_INPUT
	A : Vector_3;
	B : Vector_3;
END_VAR

V3_CROSS.X := A.Y * B.Z - A.Z * B.Y;
V3_CROSS.Y := A.Z * B.X - A.X * B.Z;
V3_CROSS.Z := A.X * B.Y - A.Y * B.X;

END_FUNCTION

// MyController/Application/cnc/vector3/V3_REV
FUNCTION V3_REV : vector_3//reverses a vector in a 3 dimensional space
VAR_INPUT
	A : Vector_3;
END_VAR

V3_REV.X := -A.X;
V3_REV.Y := -A.Y;
V3_REV.Z := -A.Z;

END_FUNCTION

// MyController/Application/cnc/vector3/V3_XANG
FUNCTION V3_XANG : LREAL//calculates the angle between the X-axis and a vectors in a 3 dimensional space
VAR_INPUT
	A : Vector_3;
END_VAR
VAR
	la: LREAL;
END_VAR

la := V3_ABS(a);
IF la > 0.0 THEN
	V3_XANG := ACOS(A.X / la);
END_IF;

END_FUNCTION

// MyController/Application/cnc/vector3/V3_YANG
FUNCTION V3_YANG : LREAL
VAR_INPUT
	A : Vector_3;//calculates the angle between the Y-axis and a vectors in a 3 dimensional space
END_VAR
VAR
	la: LREAL;
END_VAR

la := V3_ABS(a);
IF la > 0.0 THEN
	V3_YANG := ACOS(A.Y / la);
END_IF;

END_FUNCTION

// MyController/Application/cnc/vector3/V3_ZANG
FUNCTION V3_ZANG : LREAL//calculates the angle between the Z-axis and a vectors in a 3 dimensional space
VAR_INPUT
	A : Vector_3;
END_VAR
VAR
	la: LREAL;
END_VAR

la := V3_ABS(a);
IF la > 0.0 THEN
	V3_ZANG := ACOS(A.Z / la);
END_IF;

END_FUNCTION

// MyController/Application/cnc/vector3/V3_COPY
FUNCTION V3_COPY : vector_3
VAR_INPUT
	A : Vector_3;
END_VAR
VAR
END_VAR

V3_COPY.x:=A.x;
V3_COPY.y:=A.y;
V3_COPY.z:=A.z;

END_FUNCTION

// MyController/Application/cnc/vector3/V3_NORM
FUNCTION V3_NORM : LREAL
VAR_INPUT
	A:vector_3;
END_VAR
VAR
END_VAR

V3_NORM:=SQRT((A.x*A.x)+(A.y*A.y)*(A.z*A.z));

END_FUNCTION

// MyController/Application/cnc/vector3/V3_SDIV
FUNCTION V3_SDIV : vector_3//multiplies a vectors in a 3 dimensional space with a skalar M
VAR_INPUT
	A : Vector_3;
	M : LREAL;
END_VAR

V3_SDIV.X := A.X / M;
V3_SDIV.Y := A.Y / M;
V3_SDIV.Z := A.Z / M;

END_FUNCTION

// MyController/Application/cnc/vector3/V3_ADD
FUNCTION V3_ADD : vector_3
VAR_INPUT
	A : Vector_3;
	B : Vector_3;
END_VAR

V3_ADD.X := A.X + B.X;
V3_ADD.Y := A.Y + B.Y;
V3_ADD.Z := A.Z + B.Z;

END_FUNCTION

// MyController/Application/new/sc_parser
FUNCTION_BLOCK sc_parser
VAR_INPUT
END_VAR
VAR_OUTPUT
END_VAR
VAR
	error_on_line:UDINT;
	syntax_error:BOOL;
END_VAR

METHOD PRIVATE arc_lenght : LREAL
VAR_INPUT
	p1:sc_pnt;//! start position
	p2:sc_pnt;//! end position 
	center:sc_pnt;//! center IJK
	arc_radius:REFERENCE TO LREAL;//! radius result
END_VAR
VAR
	radius:LREAL;
	circumference:LREAL;
	startingAngle,endingAngle:LREAL;
	chordSquared,tau,chordHeight:LREAL;
	theta:LREAL;
END_VAR
// add center offset IJ
center.x:=center.x+p1.x;
center.y:=center.y+p1.y;
// Compute geometry.
radius:=SQRT(EXPT(center.x-p1.x,2)+EXPT(center.y-p1.y,2)); 
circumference:=2.0*M_PI*radius;
startingAngle:=math.atan2(p1.y-center.y,p1.x-center.x);
endingAngle:=math.atan2(p2.y-center.y,p2.x-center.x);

// Compute chord height of arc.
chordSquared:=SQRT(EXPT(p2.x-p1.x,2)+EXPT(p2.y-p1.y,2));
tau:= (EXPT(radius,2)-(chordSquared/4));
chordHeight := radius - tau;

// Compute angle between lines.
theta:=endingAngle-startingAngle;
	//COUNTERCLOCKWISE
	IF (theta < 0)THEN
		theta:=theta+2*M_PI;
	END_IF
 
	//CLOCKWISE
	IF (theta >= 0)THEN	
		theta:=theta-2*M_PI;;
	END_IF


arc_lenght:=ABS(circumference*(theta/(2*M_PI)));
arc_radius:=radius;
END_METHOD

METHOD PRIVATE line_lenght : LREAL
VAR_INPUT
	p0,p1:sc_pnt;
END_VAR
line_lenght:=sqrt(expt(p1.x-p0.x,2)+expt(p1.y-p0.y,2)+expt(p1.z-p0.z,2));
END_METHOD

METHOD PRIVATE sc_char_is_letter : BOOL //return true if char on pos is letter
VAR_INPUT
	str : REFERENCE TO STRING(250);
	p:INT;
END_VAR
VAR
	pt : POINTER TO ARRAY[1..255] OF BYTE;
	X: BYTE;
END_VAR
pt := ADR(str);
X := pt^[p];

IF(X>64 AND X<91) THEN
	sc_char_is_letter:= TRUE;
ELSE
	sc_char_is_letter:= FALSE;
END_IF;
END_METHOD

METHOD PRIVATE sc_findp : int
VAR_INPUT
	str : STRING(250);
	src : STRING(250);
	p: INT;
END_VAR
VAR
	i: INT;
	ls: INT;
	lx: INT;
	stp: INT;
END_VAR
ls := LEN(str);
lx := LEN(src);
IF ls < lx OR lx = 0 THEN RETURN; END_IF;
stp := ls - lx + 1;
FOR i := MAX(p,1) TO stp DO
	IF MID(str,lx,i) = src THEN
		sc_findp := i;
		RETURN;
	END_IF;
END_FOR;
sc_findp := 0;
END_METHOD

METHOD PRIVATE sc_find_nonum : int
VAR_INPUT
	str : STRING(250);
	p : INT;
END_VAR
VAR
	i: INT;
	pt : POINTER TO ARRAY[1..255] OF BYTE;
	end: INT;
	X: BYTE;
END_VAR
pt := ADR(str);
end := LEN(str);
FOR i := MAX(p,1) TO end DO;
	X := pt^[i];
	IF (X < 48 AND X <> 46 AND X <> 45) OR X > 57 THEN
		sc_find_nonum := i;
		RETURN;
	END_IF;
END_FOR;
sc_find_nonum := 0;
END_METHOD

METHOD PRIVATE sc_find_num : int
VAR_INPUT
	str : STRING(250);
	p : INT;
END_VAR
VAR
	i : INT;
	pt : POINTER TO ARRAY[1..255] OF BYTE;
	stop : INT;
	X: BYTE;
END_VAR
pt := ADR(str);
stop := LEN(str);
FOR i := MAX(p,1) TO stop DO;
	X := pt^[i];
	IF (X > 47 AND X < 58) OR X = 46 OR X = 45 THEN
		sc_find_num := i;
		RETURN;
	END_IF;
END_FOR;
sc_find_num := 0;
END_METHOD

METHOD PRIVATE sc_get_letter : INT
VAR_INPUT
	str : REFERENCE TO STRING(250);//input string
	p : INT;//start position search value
	next_ptr:REFERENCE TO INT;//result line_pointer for next value search
END_VAR
VAR
	pt : POINTER TO ARRAY[1..255] OF BYTE;
	X: BYTE;
END_VAR
pt := ADR(str);
X := pt^[p];

IF(X>64 AND X<91) THEN
	sc_get_letter:=X;
ELSE
	sc_get_letter:=0;
END_IF;
next_ptr:=p+1;
END_METHOD

METHOD PRIVATE sc_get_value : LREAL
VAR_INPUT
	str : REFERENCE TO STRING(250);//input string
	p : INT;//start position search value
	next_ptr:REFERENCE TO INT;//result line_pointer for next letter search
END_VAR
VAR
	number_start: INT;
	letter_pos: INT;
	number_end: INT;
END_VAR
number_start:=sc_find_num(str,p);	
number_end:=sc_find_nonum(str,p);
IF(number_end=0)THEN
	number_end:=LEN(str)+1;
END_IF

sc_get_value:=STRING_TO_LREAL(MID(str,number_end-number_start,number_start));
//sc_get_value:=round(sc_get_value,DECIMALS);
next_ptr:=number_end;
END_METHOD

METHOD PRIVATE sc_parse_clean : BOOL
VAR_INPUT
	plv:REFERENCE TO sc_segment;
	parsed_vec:REFERENCE TO vector_sc_segment;
END_VAR
//init parser last value, position tool ecc...
MEMUtils.MemSet(ADR(plv),0,SIZEOF(plv));
//init buffer 
parsed_vec.clear();

error_on_line:=0;	
syntax_error:=FALSE;
END_METHOD

METHOD PRIVATE sc_parse_line:UDINT
VAR_INPUT
	line:STRING(250);//line to parse
	plv:REFERENCE TO sc_segment;//parse last value store
	parsed_vec:REFERENCE TO vector_sc_segment;
	xyz:sc_pnt;//current xyz point
	set_start_on_current_position:REFERENCE TO BOOL;
	limits:cn_limits;
END_VAR
VAR
	letter:ascii_letters;
	value:LREAL;
	char_ptr:INT;
	arc_radius:LREAL;
	p_block:sc_segment;// temp block for parsing
	
	
END_VAR
//init block
MEMUtils.MemSet(ADR(p_block),0,SIZEOF(p_block));

//uppercase
line:=uppercase(line);
//remove white space
line:=trim(line);

//start from 1 char of string
char_ptr:=1;
//check letter -> value
WHILE  sc_char_is_letter(line,char_ptr) DO		
	letter:=sc_get_letter(line,char_ptr,char_ptr);	
	CASE letter OF		
		G_:		
			value:=sc_get_value(line,char_ptr,char_ptr);			
			CASE LREAL_TO_INT(value) OF				
				0://rapid move
					p_block.primitive_id:=sc_primitive_id.rapid;		
				1://feed move
					p_block.primitive_id:=sc_primitive_id.line;		
				2://arc cw move
					p_block.primitive_id:=sc_primitive_id.arc_cw;
				3://arc ccw move
					p_block.primitive_id:=sc_primitive_id.arc_ccw;			
				4://dwell
								
				16://ijk plane
										
				17://xy plane
										
				18://zx plane
										
				19://yz plane
				
				43://tool compensation on

				49://tool compensation off
				
				90://absolute coord
					plv.abs_inc:=0;				
				91://relative coord
					plv.abs_inc:=1;
			END_CASE		
		X_:
			IF(plv.abs_inc=0)THEN				
				p_block.pnt_e.x:=sc_get_value(line,char_ptr,char_ptr);	
			ELSE
				p_block.pnt_e.x:=plv.pnt_e.x+sc_get_value(line,char_ptr,char_ptr);	
			END_IF									
		Y_:
			IF(plv.abs_inc=0)THEN				
				p_block.pnt_e.y:=sc_get_value(line,char_ptr,char_ptr);	
			ELSE
				p_block.pnt_e.y:=plv.pnt_e.y+sc_get_value(line,char_ptr,char_ptr);	
			END_IF																	
		Z_:
			IF(plv.abs_inc=0)THEN				
				p_block.pnt_e.z:=sc_get_value(line,char_ptr,char_ptr);	
			ELSE
				p_block.pnt_e.z:=plv.pnt_e.z+sc_get_value(line,char_ptr,char_ptr);	
			END_IF															
		A_:
			IF(plv.abs_inc=0)THEN				
				p_block.dir_e.a:=sc_get_value(line,char_ptr,char_ptr);	
			ELSE
				p_block.dir_e.a:=plv.dir_e.a+sc_get_value(line,char_ptr,char_ptr);	
			END_IF	
		B_:
			IF(plv.abs_inc=0)THEN				
				p_block.dir_e.b:=sc_get_value(line,char_ptr,char_ptr);	
			ELSE
				p_block.dir_e.b:=plv.dir_e.b+sc_get_value(line,char_ptr,char_ptr);	
			END_IF	
		C_:
			IF(plv.abs_inc=0)THEN				
				p_block.dir_e.c:=sc_get_value(line,char_ptr,char_ptr);	
			ELSE
				p_block.dir_e.c:=plv.dir_e.c+sc_get_value(line,char_ptr,char_ptr);	
			END_IF	
		U_:
			IF(plv.abs_inc=0)THEN				
				p_block.ext_e.u:=sc_get_value(line,char_ptr,char_ptr);	
			ELSE
				p_block.ext_e.u:=plv.ext_e.u+sc_get_value(line,char_ptr,char_ptr);	
			END_IF
		V_:
			IF(plv.abs_inc=0)THEN				
				p_block.ext_e.v:=sc_get_value(line,char_ptr,char_ptr);	
			ELSE
				p_block.ext_e.v:=plv.ext_e.v+sc_get_value(line,char_ptr,char_ptr);	
			END_IF
		W_:
			IF(plv.abs_inc=0)THEN				
				p_block.ext_e.w:=sc_get_value(line,char_ptr,char_ptr);	
			ELSE
				p_block.ext_e.w:=plv.ext_e.w+sc_get_value(line,char_ptr,char_ptr);	
			END_IF
		I_:
			p_block.pnt_c.x:=sc_get_value(line,char_ptr,char_ptr);		
		J_:
			p_block.pnt_c.y:=sc_get_value(line,char_ptr,char_ptr);	
		K_:
			p_block.pnt_c.z:=sc_get_value(line,char_ptr,char_ptr);	
		F_:
			plv.vel_max:=sc_get_value(line,char_ptr,char_ptr);	
		S_:
			plv.s_value:=LREAL_TO_UINT(sc_get_value(line,char_ptr,char_ptr));
		M_:
			value:=sc_get_value(line,char_ptr,char_ptr);			
			CASE LREAL_TO_INT(value) OF
				3://spindle cw
					plv.s_dir:=TRUE;
				4://spindle ccw
					plv.s_dir:=FALSE;
			END_CASE			
			p_block.m_value:=LREAL_TO_UINT(value);
		P_:
			p_block.p_value:=LREAL_TO_UINT(sc_get_value(line,char_ptr,char_ptr));
		T_:
			plv.t_value:=LREAL_TO_UINT(sc_get_value(line,char_ptr,char_ptr));
		H_:
			plv.h_value:=LREAL_TO_UINT(sc_get_value(line,char_ptr,char_ptr));
	END_CASE		
END_WHILE


//set start position from previous line end position
IF(p_block.primitive_id <> sc_primitive_id.empty)THEN
	
	IF(set_start_on_current_position)THEN
		set_start_on_current_position:=FALSE;		
		plv.pnt_s.x:=xyz.x;
		plv.pnt_s.y:=xyz.y;
		plv.pnt_s.z:=xyz.z;
	END_IF

	//update block start positions
	p_block.pnt_s:=plv.pnt_s;
	p_block.dir_s:=plv.dir_s;
	p_block.ext_s:=plv.ext_s;
	//line  
	IF(p_block.primitive_id=sc_primitive_id.line OR p_block.primitive_id=sc_primitive_id.rapid)THEN
		p_block.path_lenght:=line_lenght(p_block.pnt_s,p_block.pnt_e);
	//arc 
	ELSIF(p_block.primitive_id=sc_primitive_id.arc_ccw OR p_block.primitive_id=sc_primitive_id.arc_cw)THEN
		p_block.path_lenght:=arc_lenght(p_block.pnt_s,p_block.pnt_e,p_block.pnt_c,arc_radius);
		p_block.radius:=arc_radius;		
	END_IF
	//update last position on plv
	plv.pnt_s:=p_block.pnt_e;
	plv.dir_s:=p_block.dir_e;
	plv.ext_s:=p_block.ext_e;
ELSE
	p_block.pnt_s:=plv.pnt_s;
	p_block.dir_s:=plv.dir_s;
	p_block.ext_s:=plv.ext_s;
END_IF

p_block.traject_lenght_end:=p_block.path_lenght+plv.traject_lenght_end;
p_block.traject_lenght_begin:=p_block.traject_lenght_end-p_block.path_lenght;

//update trajectory lenght on plv
plv.traject_lenght_end:=p_block.traject_lenght_end;

//update block
IF(p_block.primitive_id=sc_primitive_id.rapid)THEN
	p_block.vel_max:=limits.max_vel;
ELSE
	p_block.vel_max:=plv.vel_max;
END_IF

IF(p_block.vel_max>limits.max_vel)THEN
	p_block.vel_max:=limits.max_vel;
END_IF
p_block.pnt_e:=plv.pnt_s;
p_block.dir_e:=plv.dir_s;
p_block.ext_e:=plv.ext_s;
p_block.s_value:=plv.s_value;
p_block.s_dir:=plv.s_dir;
p_block.t_value:=plv.t_value;
p_block.h_value:=plv.h_value;
p_block.gcode_line_nr:=plv.gcode_line_nr;
plv.gcode_line_nr:=plv.gcode_line_nr+1;

//add line to motion block buffer
parsed_vec.push_back(p_block);
END_METHOD

METHOD PRIVATE sc_parse_start : BOOL
VAR_INPUT
	gcode_lines:REFERENCE TO ARRAY[0..MAX_GCODE_LINE]OF STRING(250);
	plv:REFERENCE TO sc_segment;//parse last value store
	parsed_vec:REFERENCE TO vector_sc_segment;
	xyz:sc_pnt;//current xyz point
	set_start_on_current_position:BOOL;
	limits:cn_limits;
END_VAR
VAR
	i:UDINT;
	temp_line:STRING(250);
	comm_start:INT;
	comm_end:INT;
END_VAR
FOR i:=0 TO MAX_GCODE_LINE DO	
	//copy input string to temp
	temp_line:=gcode_lines[i];
	IF(temp_line='')THEN
		EXIT;
	END_IF;
	//find start comment <-
	comm_start:=sc_findp(temp_line,'(',1);
	IF(comm_start<>0)THEN
		i:=i+1;
		//jump comment line
		temp_line:=gcode_lines[i];
	END_IF	
	//parse line
	error_on_line:=sc_parse_line(temp_line,plv,parsed_vec,xyz,set_start_on_current_position,limits);
	IF(UDINT_TO_BOOL(error_on_line))THEN
		syntax_error:=TRUE;
		EXIT;
	END_IF								
END_FOR
END_METHOD

METHOD PRIVATE to_upper : byte
VAR_INPUT
	IN : BYTE;
END_VAR
IF in > 96 AND in < 123 THEN
   TO_UPPER := in AND 16#DF;
ELSIF in > 223 AND in <> 247 AND in <> 255  THEN
   TO_UPPER := in AND 16#DF;
ELSE
   TO_UPPER := in;
END_IF;
END_METHOD

METHOD PRIVATE trim : string
VAR_INPUT
	str : STRING(250);
END_VAR
VAR
	p: INT;
END_VAR
TRIM := str;
REPEAT
	p := FIND(trim,' ');
	IF p > 0 THEN TRIM := REPLACE(TRIM,'',1,p); END_IF;
UNTIL p = 0	END_REPEAT;
END_METHOD

METHOD PRIVATE uppercase : STRING
VAR_INPUT
	str : STRING(250);
END_VAR
VAR
	pt : POINTER TO BYTE;
	p: INT;
	l: INT;
END_VAR
pt := ADR(UPPERCASE);
UPPERCASE := str;
l := LEN(str);
FOR p := 1 TO l DO
	pt^ := TO_UPPER(pt^);
	pt := pt + 1;
END_FOR;
END_METHOD

END_FUNCTION_BLOCK

// MyController/Application/new/sc_optimizer
FUNCTION_BLOCK sc_optimizer
VAR_INPUT
END_VAR
VAR_OUTPUT
END_VAR
VAR
END_VAR

METHOD arc_arc_angle : bool
VAR_INPUT
	p0:sc_pnt;
	p1:sc_pnt;
	p2:sc_pnt;
	p3:sc_pnt;
	p4:sc_pnt;
	angle_deg:REFERENCE TO LREAL;
END_VAR
VAR
	pi0,pi1:sc_pnt;
	
END_VAR
interpolate_arc(p0,p1,p2,0.9,pi0);
interpolate_arc(p2,p3,p4,0.1,pi1);
line_line_angle(pi0,p2,pi1,angle_deg);
END_METHOD

METHOD arc_line_angle : bool
VAR_INPUT
	p0:sc_pnt;
	p1:sc_pnt;
	p2:sc_pnt;
	p3:sc_pnt;
	angle_deg:REFERENCE TO LREAL;
END_VAR
VAR
	pi:sc_pnt;

END_VAR
interpolate_arc(p0,p1,p2,0.9,pi);
line_line_angle(pi,p2,p3,angle_deg);
END_METHOD

METHOD get_blockangles : BOOL
VAR_INPUT
	blockvec:REFERENCE TO vector_sc_segment;
	start:REFERENCE TO UDINT;
	end:REFERENCE TO UDINT;
END_VAR
VAR	
	i: UDINT;
	angle_deg:LREAL;
END_VAR
IF(blockvec.size()>0)THEN //! Vector safe.}
	
	FOR i:=start TO end-1 DO
		
		IF(blockvec.data[i].primitive_id=sc_primitive_id.line AND  blockvec.data[i+1].primitive_id=sc_primitive_id.line)THEN
			line_line_angle(blockvec.data[i].pnt_s,blockvec.data[i].pnt_e,blockvec.data[i+1].pnt_e,angle_deg);
			blockvec.data[i].angle_end:=angle_deg;
		END_IF
		
		IF(blockvec.data[i].primitive_id=sc_primitive_id.line AND (blockvec.data[i+1].primitive_id=sc_primitive_id.arc_ccw OR blockvec.data[i+1].primitive_id=sc_primitive_id.arc_cw))THEN
			line_arc_angle(blockvec.data[i].pnt_s,blockvec.data[i].pnt_e,blockvec.data[i+1].pnt_c,blockvec.data[i+1].pnt_e,angle_deg);
			blockvec.data[i].angle_end:=angle_deg;
		END_IF
		
		IF((blockvec.data[i].primitive_id=sc_primitive_id.arc_ccw OR blockvec.data[i].primitive_id=sc_primitive_id.arc_cw) AND blockvec.data[i+1].primitive_id=sc_primitive_id.line)THEN
			arc_line_angle(blockvec.data[i].pnt_s,blockvec.data[i].pnt_c,blockvec.data[i].pnt_e,blockvec.data[i+1].pnt_e,angle_deg);
			blockvec.data[i].angle_end:=angle_deg;
		END_IF
		
		IF((blockvec.data[i].primitive_id=sc_primitive_id.arc_ccw OR blockvec.data[i].primitive_id=sc_primitive_id.arc_cw) AND (blockvec.data[i+1].primitive_id=sc_primitive_id.arc_ccw OR blockvec.data[i+1].primitive_id=sc_primitive_id.arc_cw))THEN
			arc_arc_angle(blockvec.data[i].pnt_s,blockvec.data[i].pnt_c,blockvec.data[i].pnt_e,blockvec.data[i+1].pnt_c,blockvec.data[i+1].pnt_e,angle_deg);
			blockvec.data[i].angle_end:=angle_deg;
		END_IF
	END_FOR
END_IF
END_METHOD

METHOD get_corner_ve_blockangles : BOOL
VAR_INPUT
	blockvec:REFERENCE TO vector_sc_segment;
	start:REFERENCE TO UDINT;
	end:REFERENCE TO UDINT;
END_VAR
VAR	
	i: UDINT;
	angle_deg,factor,ve:LREAL;
END_VAR
IF(blockvec.size()<>0)THEN
	FOR i:=start TO  end-1 DO
		
		IF(blockvec.data[i].angle_end<=STOP_ANGLE)THEN //! Stop required.
			blockvec.data[i].vel_end:=0;
			//! Set next block vo to zero.
			IF(i<blockvec.size()-1)THEN
				blockvec.data[i+1].vel_start:=0;
			END_IF
		END_IF
	
		IF(blockvec.data[i].angle_end>STOP_ANGLE)THEN //! Percentage ve up to 180 degrees. //! 180 degrees = colinear.
			angle_deg:=blockvec.data[i].angle_end;
			factor:=(angle_deg-STOP_ANGLE)/STOP_ANGLE; //! 0-1, 1=straight on. 0=90 degrees.
			ve:=blockvec.data[i].vel_max*factor*ANGLE_VEL_FACTOR;
	
			blockvec.data[i].vel_end:=ve;
			//! Set next block vo to this ve.
			IF(i<blockvec.size()-1)THEN
				blockvec.data[i+1].vel_start:=ve;
			END_IF
		END_IF
		
	END_FOR
END_IF
END_METHOD

METHOD get_velmax_gforce : bool
VAR_INPUT
	blockvec:REFERENCE TO vector_sc_segment;
	gforcemax:LREAL;
	start:REFERENCE TO UDINT;
	end:REFERENCE TO UDINT;
END_VAR
VAR
	i:UDINT;
	radius,gforce,maxvel_arc:LREAL;
	vm:LREAL;
END_VAR
IF(blockvec.size()<>0)THEN
	FOR i:=start TO end-1 DO
		IF(blockvec.data[i].primitive_id=sc_primitive_id.arc_cw OR blockvec.data[i].primitive_id=sc_primitive_id.arc_ccw)THEN	
			
			radius:=blockvec.data[i].radius;	
			
			//! Checks gforce using the program's velmax value.	
			vm:=blockvec.data[i].vel_max;							
			sc_get_gforce(vm,radius,gforce);
	
			IF(gforce>gforcemax)THEN
				maxvel_arc:=0;
				sc_set_gforce(radius,gforcemax,maxvel_arc);
				blockvec.data[i].vel_max:=maxvel_arc;
			END_IF			
		END_IF
	END_FOR
END_IF
END_METHOD

METHOD line_arc_angle : bool
VAR_INPUT
	p0:sc_pnt;
	p1:sc_pnt;
	p2:sc_pnt;
	p3:sc_pnt;
	angle_deg:REFERENCE TO LREAL;
END_VAR
VAR
	pi:sc_pnt;
END_VAR
interpolate_arc(p1,p2,p3,0.1,pi);
line_line_angle(p0,p1,pi,angle_deg);
END_METHOD

METHOD line_line_angle : bool
VAR_INPUT
	p0:sc_pnt;
	p1:sc_pnt;
	p2:sc_pnt;
	angle_deg:REFERENCE TO LREAL;
END_VAR
VAR
	p00,p11,p22,v1,v2:Vector_3;
	dot,angle_rad:LREAL;
END_VAR
p00:=p_to_v(p0);
p11:=p_to_v(p1);
p22:=p_to_v(p2);

v1:=V3_SUB(p00,p11);
v2:=V3_SUB(p22,p11);

v1:=V3_NORMALIZED(v1);
v2:=V3_NORMALIZED(v2);

dot:=V3_DOT(v1,v2);
angle_rad:=ACOS(dot);
angle_deg:=angle_rad*to_degrees;
END_METHOD

METHOD p_to_v : Vector_3 //sc_pnt to vector3
VAR_INPUT
	in:sc_pnt;
END_VAR
p_to_v.x:=in.x;
p_to_v.y:=in.y;
p_to_v.z:=in.z;
END_METHOD

METHOD sc_get_gforce : bool
VAR_INPUT
	vel_mm_sec:LREAL;
	radius:LREAL;
	gforce:LREAL;
END_VAR
VAR	
	circumfence: LREAL;
	rps: LREAL;
	a:LREAL;
END_VAR
circumfence:=(radius*2)*M_PI;
rps:=vel_mm_sec/circumfence;
a:=4*(M_PI*M_PI)*radius*(rps*rps); //! [mm/s^2]
gforce:=a*0.0001; //! [g]
END_METHOD

METHOD sc_optimize_all : BOOL
VAR_INPUT
	blockvec:REFERENCE TO vector_sc_segment;
	line_start:UDINT;
	line_end:UDINT;
END_VAR
line_start:=LIMIT(0,line_start,blockvec.size());
line_end:=LIMIT(line_start,line_end,blockvec.size());



//! Calculate motion block corners.
get_blockangles(blockvec,line_start,line_end);

//! Set end velocity, based on block corners, if no angle, ve is set to vm at this stage.
get_corner_ve_blockangles(blockvec,line_start,line_end);

//! Set the velmax for arc's using gforce value. Set the velmax for lines to program velmax.
get_velmax_gforce(blockvec,gforcemax,line_start,line_end);

//set g0 ve vo
sc_optimize_G0_ve(blockvec,line_start,line_end);

//optimize ve <--
sc_optimize_G123_ve_backward(blockvec,line_start,line_end);

//optimize ve -->
sc_optimize_G123_ve_forward(blockvec,line_start,line_end);
END_METHOD

METHOD sc_optimize_G0_ve : BOOL
VAR_INPUT
	blockvec:REFERENCE TO vector_sc_segment;
	start:REFERENCE TO UDINT;
	end:REFERENCE TO UDINT;
END_VAR
VAR
	i:UDINT;
END_VAR
IF(blockvec.size()<>0)THEN
	FOR i:=start TO end-1 DO
	
		//! End velocity=0 if motion is G0, rapid.
		IF(blockvec.data[i].primitive_id=sc_primitive_id.rapid)THEN 
			blockvec.data[i].vel_start:=0;
			blockvec.data[i].vel_end:=0;
	
			//! Set next block vo to 0.
			IF(i<blockvec.size()-1)THEN
				blockvec.data[i+1].vel_start:=0;
			END_IF
		END_IF
	END_FOR
END_IF
END_METHOD

METHOD sc_optimize_G123_ve_backward :BOOL
VAR_INPUT
	blockvec:REFERENCE TO vector_sc_segment;
	start:REFERENCE TO UDINT;
	end:REFERENCE TO UDINT;
END_VAR
VAR
	i:UDINT;
	vo,ve,vm,tarpos:LREAL;
	r_vel,r_acc,r_pos:LREAL;
	finish:BOOL;
	p_data:sc_data;
	pcurve:sc_engine;
	j:LREAL;
	
END_VAR
IF(blockvec.size()<>0)THEN
	FOR i:=end-1 TO start+1 BY-1 DO 
		
		IF(blockvec.data[i].primitive_id<>sc_primitive_id.rapid AND blockvec.data[i].primitive_id<>sc_primitive_id.empty)THEN 
			//! Swap vo,ve.
			ve:=blockvec.data[i].vel_start;
			vo:=blockvec.data[i].vel_end;
			vm:=blockvec.data[i].vel_max;
			tarpos:=blockvec.data[i].path_lenght;	

			MEMUtils.MemSet(ADR(p_data),0,SIZEOF(p_data));
			
			pcurve.set_cycle_time(CT,p_data);
			
			finish:=FALSE;
			WHILE NOT finish DO				
				pcurve.set_data(tarpos,vo,ve,vm,limits.max_acc,limits.max_jerk,1,p_data);	
				pcurve.update(p_data,1);
				pcurve.get_result(r_pos,r_vel,r_acc,finish,p_data);			
			END_WHILE
			
			IF(ve<>0)THEN
				blockvec.data[i].vel_start:=r_vel;
				blockvec.data[i-1].vel_end:=r_vel;
			END_IF
			
			blockvec.data[i].back_optim:=TRUE;
		END_IF
	END_FOR
END_IF
END_METHOD

METHOD sc_optimize_G123_ve_forward : BOOL
VAR_INPUT
	blockvec:REFERENCE TO vector_sc_segment;
	start:REFERENCE TO UDINT;
	end:REFERENCE TO UDINT;
END_VAR
VAR
	i:UDINT;
	vo,ve,vm,tarpos:LREAL;
	r_vel,r_acc,r_pos:LREAL;
	finish:BOOL;
	p_data:sc_data;
	pcurve:sc_engine;

END_VAR
IF(blockvec.size()<>0)THEN	
	FOR i:=start TO end-1 DO 
	
		IF(blockvec.data[i].primitive_id<>sc_primitive_id.rapid AND blockvec.data[i].primitive_id<>sc_primitive_id.empty)THEN 
	
			vo:=blockvec.data[i].vel_start;
			ve:=blockvec.data[i].vel_end;
			vm:=blockvec.data[i].vel_max;
			tarpos:=blockvec.data[i].path_lenght;
			
			MEMUtils.MemSet(ADR(p_data),0,SIZEOF(p_data));
			
			pcurve.set_cycle_time(CT,p_data);
						
			finish:=FALSE;
			WHILE NOT finish DO			
				pcurve.set_data(tarpos,vo,ve,vm,limits.max_acc,limits.max_jerk,1,p_data);	
				pcurve.update(p_data,1);
				pcurve.get_result(r_pos,r_vel,r_acc,finish,p_data);
			END_WHILE
			
			IF(ve<>0)THEN
				blockvec.data[i].vel_end:=r_vel;		
				IF(i<blockvec.size()-1)THEN  
					blockvec.data[i+1].vel_start:=r_vel;
				END_IF				
			END_IF
			
			blockvec.data[i].forward_optim:=TRUE;
		END_IF
	END_FOR
END_IF
END_METHOD

METHOD sc_set_gforce : bool
VAR_INPUT
	radius:LREAL;
	gforce:LREAL;
	vel_mm_sec:reference TO LREAL;
END_VAR

VAR
	rps: LREAL;
	circumfence: LREAL;
	a:LREAL;
END_VAR
circumfence:=(radius*2)*M_PI;
a:=gforce/0.0001;
rps:= SQRT(a/(4*(M_PI*M_PI)*radius));
vel_mm_sec:=rps*circumfence;
END_METHOD

END_FUNCTION_BLOCK

// MyController/Application/Visualization
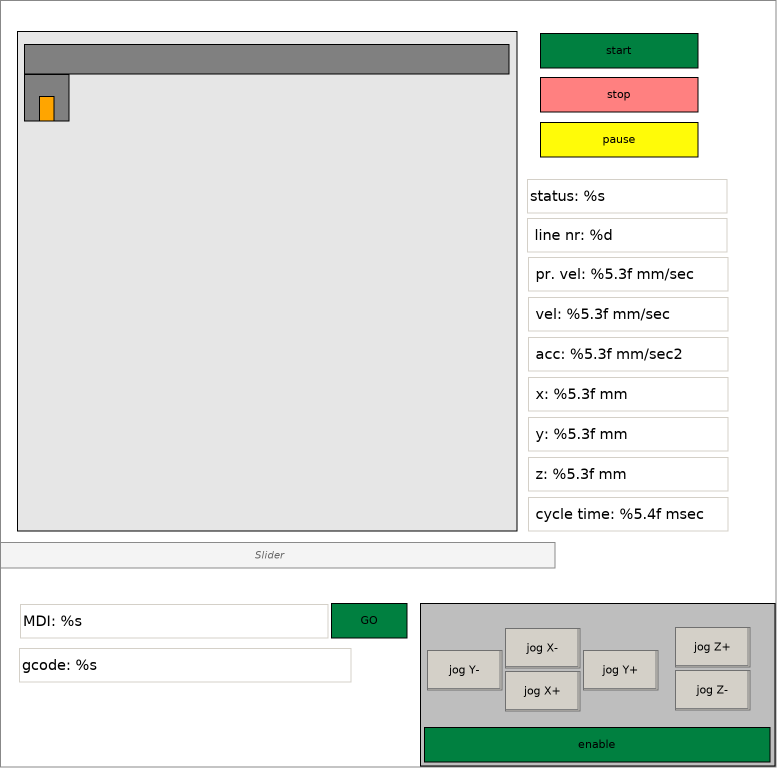
VISUALIZATION Visualization  // 777x768
    Rectangle (17,31 500x500)
    RoundedRectangle (540,33 158x35), "start"
        tap test.start
        OnMouseUp:  ToggleVariable=test.start
    Textfield (528,297 200x34), "vel: %5.3f mm/sec", text variable: test.velocity
    Textfield (528,337 200x34), "acc: %5.3f mm/sec2", text variable: test.acceleration
    Textfield (528,377 200x34), "x: %5.3f mm", text variable: test.x
    Textfield (528,417 200x34), "y: %5.3f mm", text variable: test.y
    Textfield (528,457 200x34), "z: %5.3f mm", text variable: test.z
    Textfield (528,497 200x34), "cycle time: %5.4f msec", text variable: test.performance
    RoundedRectangle (540,77 158x35), "stop"
        tap test.stop
        OnMouseUp:  ToggleVariable=test.stop
    RoundedRectangle (540,122 158x35), "pause"
        toggle test.pause
    Rectangle (24,44 485x30)
        p2773130477: test.y
        p1126004900: test.y
    Textfield (527,218 200x34), "line nr: %d", text variable: test.line_nr
    Rectangle (24,74 45x47)
        p3528305787: test.x
        p874137650: test.x
        p2773130477: test.y
        p1126004900: test.y
    Rectangle (39,96 15x25)
        p3528305787: test.x
        p874137650: test.x
        p2773130477: test.y-test.z
        p1126004900: test.y-test.z
    Textfield (528,257 200x34), "pr. vel: %5.3f mm/sec", text variable: test.programmed_velocity
    Slider (-16,542 571x26), variable: test.feed_override, scale 0..100
    Textfield (527,179 200x34), "status: %s", text variable: test.state
    Textfield (20,604 308x34), "MDI: %s", text variable: test.mdi
        OnMouseClick: write the text variable via Edit
    RoundedRectangle (331,603 76x35), "GO"
        tap test.mdi_start
    Textfield (19,648 332x34), "gcode: %s", text variable: test.gcode[test.line_nr]
    Rectangle (420,603 355x163)
    Button (505,671 75x40), "jog X+"
        tap test.x_up
    Button (505,628 75x40), "jog X-"
        tap test.x_dn
    Button (583,650 75x40), "jog Y+"
        tap test.y_up
    Button (427,650 75x40), "jog Y-"
        tap test.y_dn
    Button (675,627 75x40), "jog Z+"
        tap test.z_up
    Button (675,670 75x40), "jog Z-"
        tap test.z_dn
    RoundedRectangle (424,727 346x35), "enable"
        toggle test.jog_enable
END_VISUALIZATION
